FUNCTION_BLOCK DepotControl (* Basic FB with empty ECC *)
  (* Standard: 61499-2 *)
  (* Version 1.0, 2021-09-15, dorofeev *)
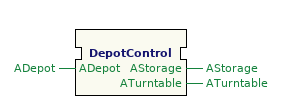
  SOCKETS
    ADepot : ADepot;
  END_SOCKETS
  PLUGS
    AStorage : AStorage;
    ATurntable : ATurntable;
  END_PLUGS
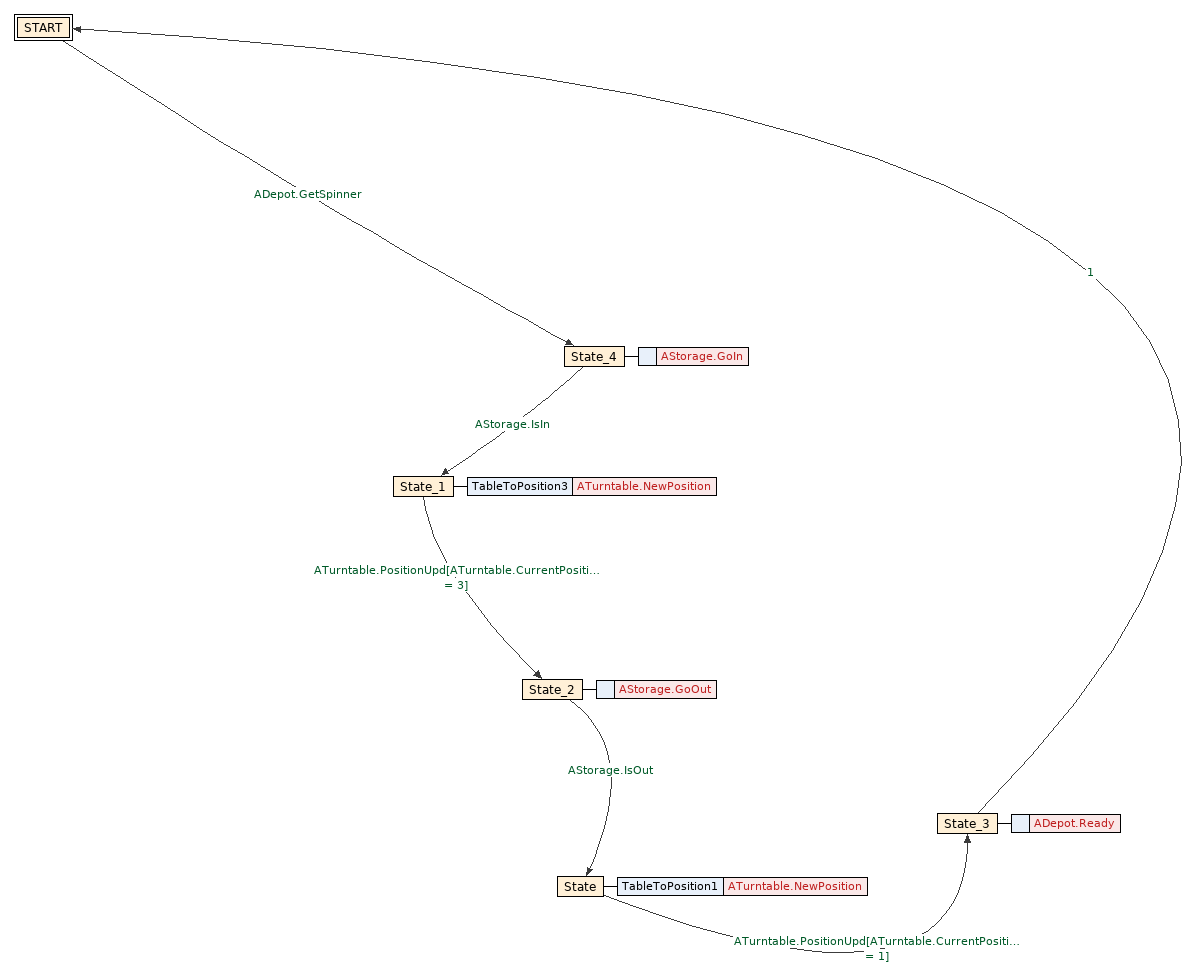
  EC_STATES
    START; (* Initial State *)
    State_1 : TableToPosition3 -> ATurntable.NewPosition;
    State_2 : -> AStorage.GoOut;
    State_3 : -> ADepot.Ready;
    State_4 : -> AStorage.GoIn;
    State : TableToPosition1 -> ATurntable.NewPosition;
  END_STATES
  EC_TRANSITIONS
    State_1 TO State_2 := ATurntable.PositionUpd[ATurntable.CurrentPosition = 3];
    State_4 TO State_1 := AStorage.IsIn;
    START TO State_4 := ADepot.GetSpinner;
    State_3 TO START := 1;
    State_2 TO State := AStorage.IsOut;
    State TO State_3 := ATurntable.PositionUpd[ATurntable.CurrentPosition = 1];
  END_TRANSITIONS
  ALGORITHM TableToPosition3 IN ST: (* New Algorithm *)
ATurntable.Position := 3;
  END_ALGORITHM
  ALGORITHM TableToPosition1 IN ST: (* New Algorithm *)
ATurntable.Position := 1;
  END_ALGORITHM
END_FUNCTION_BLOCK
